FUNCTION_BLOCK FB_Persistent

(********************************************************************************************************)
(*								Beckhoff Automation Poland												*)
(* 									FB_Persistent 	v1.5												*)
(* 										20.08.2014														*)
(* 							v1.5 - zmiana minimalnego interwalu zapisu									*)
(* 					Blok funkcyjny zapisujący zmienne typu persistent na karcie CF						*)
(* 						Możliwy zapis na żądanie lub z określoną częstotliwością.  						*)
(* 				Pozostawienie wejscia tInterval bez zmiennej wyłacza funkcję zapisu cyklicznego			*)
(* 							Minimalny czas między zapisem cyklicznym 30s								*)
(* 				Konieczne jest dodanie biblioteki TcUtilities.lib, TcSystem.lib oraz TcBase.lib			*)
(*			 UWAGA: Blok przygotowany dla RunTime 1 port 851 - typowa konfiguracja 						*)
(*______________________________________________________________________________________________________*)

VAR_INPUT
	bWrite					: BOOL;						(*Zapis na rozkaz *)
	tInterval				: TIME:=T#71582M47S295MS;	(*Czestotliwosc zapisu na karte CF*)
END_VAR
VAR_OUTPUT
	bBusy					: BOOL;
	bErr					: BOOL;
	udErrID					: UDINT;
END_VAR
VAR
	fbWritePersistentData	: FB_WritePersistentData; 	(* Blok zapisu *)
	t1						: TON;						(* Timer zapisu *)
	_GETCURTASKINDEX		: GETCURTASKINDEX;			(* Informacja o Tasku *)
	BIndex					: BYTE;						(* Nr tasku *)
END_VAR

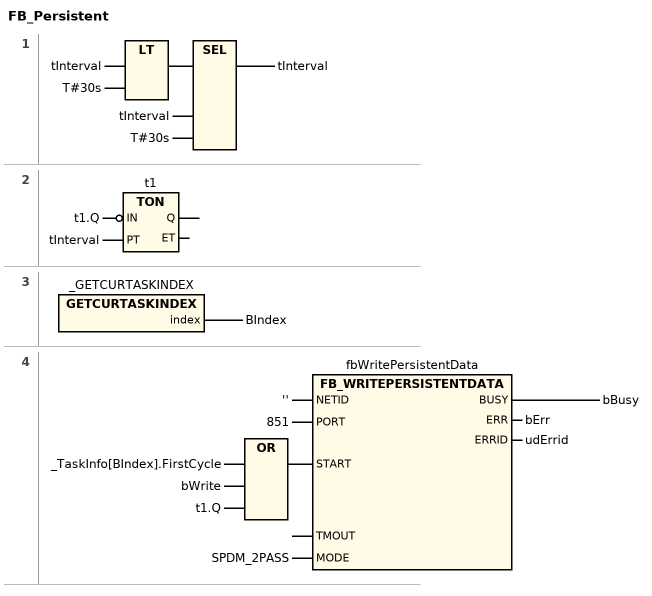
// NETWORK 1
tInterval := SEL(tInterval < T#30s, tInterval, T#30s);

// NETWORK 2
t1(IN := NOT t1.Q, PT := tInterval); // TON

// NETWORK 3
_GETCURTASKINDEX(); // GETCURTASKINDEX
BIndex := _GETCURTASKINDEX.index;

// NETWORK 4
fbWritePersistentData(
    NETID := '',
    PORT := 851,
    START := _TaskInfo[BIndex].FirstCycle OR bWrite OR t1.Q,
    MODE := SPDM_2PASS,
    ERR => bErr,
    ERRID => udErrid); // FB_WRITEPERSISTENTDATA
bBusy := fbWritePersistentData.BUSY;

END_FUNCTION_BLOCK

(* stored: Version 1.1.0.1, ProductVersion 3.1.4026.13, FileIdentifier 695c9ecc75ee8f48c72be406076b89964e6f61fd, FileSignature a6c763218445610413075f1874032825f26b942bbd205ada03c3473ff626c4ce1e99e6e2192f91a4adcfe35d9c12610ee732dbee85f7b4b3c7f9e8d409b282b5458be2a9168417ba3be9ee6ae0cc5808d3feb15ea6a415d8fd630e1a76c2c4d9b2560f3c59a0b367ec5797e14a9b75ba3066816aac994c96c86dc5c2baad52b6def3a49226feacc633834fc1d51aecf3dde3fc6f17965c1dba355984f02896b1363c2f2743f2cf4a17e2f7bbf8647abbef8d79a83d086a9983ef0f0ea24d726d9017c52f9d08e2cfc6506d2e90c22a210024e4722162c2d5cc471405dc8b681cdcf75fa03a5a8f8c028d461661ecfa640d2ecbfe2084e5f14a892bdd366c20df
   POU FB_Persistent: Id {040600c4-f85f-45bb-b3dd-9c0bbbb5e071}, SpecialFunc None *)
